// Mitsubishi GX Works2 project: ZhaoQing_HuaCheng2_1.1修改   PLC: Q03UDE
// 化成线2号柜

TYPE BarCylinderIO : STRUCT
  xPresentSwitch : BOOL;  (* 行程开关 *)
  xBarCylinder : BOOL;  (* 阻挡气缸 *)
  xEmpty : BOOL;  (* 为空指示 *)
  xTransportMotorCW : BOOL;  (* 输送电机正转 *)
  tLeaveDelay : TIME;  (* 放行延时 *)
  xUnload : BOOL;  (* 下料 *)
  xBarCylinderButton : BOOL;  (* 阻挡气缸 *)
  xTransportMotorCWButton : BOOL;  (* 输送电机正转按钮 *)
  xLoad : BOOL;  (* 上料 *)
  xNextRun : BOOL;  (* 下位设备开始运行 *)
  xTransportMotorCCWButton : BOOL;  (* 输送电机反转按钮 *)
  xTransportMotorCCW : BOOL;  (* 输送电机反转 *)
END_STRUCT END_TYPE

TYPE ConveyorIO : STRUCT
  xCWPresent : BOOL;  (* 正转检测有无传感器 *)
  xCCWPresent : BOOL;  (* 反转检测有无传感器 *)
  xLoad : BOOL;  (* 上料请求 *)
  xUnload : BOOL;  (* 下料请求 *)
  xMotorCW : BOOL;  (* 电机正转 *)
  xMotorCCW : BOOL;  (* 电机反转 *)
  xEmpty : BOOL;  (* 线体状态为空 *)
  xNextRun : BOOL;  (* 下段线体运行 *)
  xUnloadCCW : BOOL;  (* 下料为反转 *)
  xloadCCW : BOOL;  (* 上料为反转 *)
  xLeave : BOOL;  (* 已经离开 *)
  xForward : BOOL;  (* 正转手动 *)
  xBackward : BOOL;  (* 反转手动 *)
  xBusy : BOOL;  (* 工作中 *)
  tLeaveDelay : TIME;  (* 离开延时设置 *)
  xPutInto : BOOL;  (* 线体直接投入物料 *)
  xLoadAlarrm : BOOL;  (* 上料报警 *)
  xUnloadAlarm : BOOL;  (* 下料报警 *)
  tLoadDelay : TIME;  (* 进入延时设置 *)
  iProductCategory : INT;  (* 产品种类 *)
END_STRUCT END_TYPE

TYPE RGVCommunication : STRUCT
  xFullLoadRequest : BOOL;  (* 满框上料请求 *)
  xFullUnloadRequest : BOOL;  (* 满框下料请求 *)
  xEmptyLoadRequest : BOOL;  (* 空框上料请求 *)
  xEmptyUnloadRequest : BOOL;  (* 空框下料请求 *)
  xFullLoadRequestAkn : BOOL;  (* 满框上料请求确认 *)
  xFullUnloadRequestAkn : BOOL;  (* 满框下料请求确认 *)
  xEmptyLoadRequestAkn : BOOL;  (* 空框上料请求确认 *)
  xEmptyUnloadRequestAkn : BOOL;  (* 空框下料请求确认 *)
  xFullLoadComplete : BOOL;  (* 满框上料完成 *)
  xFullUnloadComplete : BOOL;  (* 满框下料完成 *)
  xEmptyLoadComplete : BOOL;  (* 空框上料完成 *)
  xEmptyUnloadComplete : BOOL;  (* 空框下料完成 *)
  xFullLoadCompleteAkn : BOOL;  (* 满框上料完成确认 *)
  xFullUnloadCompleteAkn : BOOL;  (* 满框下料完成确认 *)
  xEmptyLoadCompleteAkn : BOOL;  (* 空框上料完成确认 *)
  xEmptyUnloadCompleteAkn : BOOL;  (* 空框下料完成确认 *)
END_STRUCT END_TYPE

TYPE ShuttleCarIO : STRUCT
  xReady : BOOL;  (* 准备就绪 *)
  xForward : BOOL;  (* 正转 *)
  xBackward : BOOL;  (* 反转 *)
  iCurrentPos : INT;  (* 当前位置 *)
  iDestinationPos : INT;  (* 目标位置 *)
  xCW : BOOL;  (* 正转输出 *)
  xCCW : BOOL;  (* 反转输出 *)
  xBrake : BOOL;  (* 刹车 *)
  xHomeSwitch : BOOL;  (* 零位接近开关 *)
  xPosLimit : BOOL;  (* 正限位 *)
  xNegLimit : BOOL;  (* 负限位 *)
  xMDIExe : BOOL;  (* MDI开始 *)
  xMDIDone : BOOL;  (* MDI 完成 *)
  xPassLimit : BOOL;  (* 限位屏蔽 *)
  xPosLimitCatch : BOOL;  (* 正限位捕捉 *)
  xNegLimitCatch : BOOL;  (* 负限位捕捉 *)
  xHomeExe : BOOL;  (* 开始寻零 *)
  xHomeDone : BOOL;  (* 寻零完成 *)
  xHomeBusy : BOOL;  (* 寻零中 *)
  xHomeFailed : BOOL;  (* 寻零失败 *)
  xBusy : BOOL;  (* 工作中 *)
END_STRUCT END_TYPE

TYPE SwitchIO : STRUCT
  xLiftCylinderRetractDetect : BOOL;
  xLiftCylinderExtendDetect : BOOL;
  xLiftCylinderRetract : BOOL;
  xLiftCylinderExtend : BOOL;
  xEntryBarCylinderRetract : BOOL;
  xLiftCylinderExtendInit : BOOL;
  xEntryEnable : BOOL;
  xExitEnable : BOOL;
  xExitBarCylinderRetract : BOOL;
  xSwithEnable : BOOL;
  xLiftCylinderRetractButton : BOOL;
  xLiftCylinderExtendButton : BOOL;
  xEntryBarCylinderRetractButton : BOOL;
  xExitBarCylinderRetractButton : BOOL;
END_STRUCT END_TYPE

// global labels: Global1
VAR_GLOBAL
  g_xAuto AT M11 : BOOL;  (* 自动 *)
  g_xManual : BOOL;  (* 手动 *)
  g_xEStop AT X3 : BOOL;  (* 急停 *)
  g_xReset AT X0 : BOOL;  (* 复位 *)
  g_xStackLampRed AT Y100 : BOOL;
  g_xStackLampAmber AT Y101 : BOOL;
  g_xStackLampGreen AT Y102 : BOOL;
  g_xBuzzer AT Y103 : BOOL;
  g_xStop AT M2 : BOOL;  (* 停止 *)
  g_xLocalAutoStart AT M1 : BOOL;
  g_xRemoteAutoStart AT M0 : BOOL;
  g_xRemoteAuto AT M10 : BOOL;
  g_iState AT D40 : INT;
  g_iLocalAutoStep : INT;
  g_xError : BOOL;
  g_xStart : BOOL;  (* 启动 *)
END_VAR

// task Task_01 (event TRUE, interval 0, priority 31): Start, POU, UDP

FUNCTION_BLOCK BarCylinder
VAR_IN_OUT
  BarCylinderIO : BarCylinderIO;
END_VAR
VAR
  m_tonViaDelay : TON;  (* 卸料延时定时器 *)
  m_xViaDelay : BOOL;  (* 通过延时 *)
  m_tViaDelayElapse : TIME;  (* 通过延时当前时间 *)
  m_xInitial : BOOL;  (* 初始化 *)
END_VAR
  (***********************************************************************
阻挡器模块，
由一个行程开关，一个阻挡器，一个倍速链输送电机组成
具有手动与自动模式
xEmpty显示当前为空料的状态
xUnload为卸料信号，连接下一设备的xEmpty信号
*************************************************************************)

  (*初始化，离开延时时间设置为5秒*)
IF NOT m_xInitial THEN
	 BarCylinderIO.tLeaveDelay :=T#5s;
	m_xInitial:=1;
END_IF;
IF g_xManual THEN    (*手动*)
	BarCylinderIO.xNextRun:=0;
	IF BarCylinderIO.xBarCylinderButton THEN
		BarCylinderIO.xBarCylinder:=1;
	ELSE
		BarCylinderIO.xBarCylinder:=0;
	END_IF;
	IF BarCylinderIO.xTransportMotorCWButton 
		AND NOT BarCylinderIO.xTransportMotorCCWButton 
		AND NOT BarCylinderIO.xTransportMotorCCW   THEN
		BarCylinderIO.xTransportMotorCW:=1;
	ELSE
		BarCylinderIO.xTransportMotorCW:=0;
	END_IF;
	IF BarCylinderIO.xTransportMotorCCWButton 
		AND NOT BarCylinderIO.xTransportMotorCWButton 
		AND NOT BarCylinderIO.xTransportMotorCW   THEN
		BarCylinderIO.xTransportMotorCCW:=1;
	ELSE
		BarCylinderIO.xTransportMotorCCW:=0;
	END_IF;
END_IF;
(*离开延时定时器*)
m_tonViaDelay(IN:=NOT  BarCylinderIO.xPresentSwitch AND g_xAuto  ,PT:= BarCylinderIO.tLeaveDelay ,Q:= BarCylinderIO.xEmpty ,ET:=m_tViaDelayElapse );

IF g_xAuto THEN(*自动*)
    IF BarCylinderIO.xUnload  AND NOT BarCylinderIO.xEmpty AND NOT BarCylinderIO.xNextRun THEN(*收到卸料命令，当阻挡器不为空时*)
    	BarCylinderIO.xBarCylinder:=1;
    	BarCylinderIO.xNextRun:=1;(*确保下料命令只执行一次，防止物料在输送过程中又有卸料命令导致多事卸料*)
    	BarCylinderIO.xTransportMotorCW:=1;
    END_IF;
    IF NOT  BarCylinderIO.xUnload  THEN
    	BarCylinderIO.xNextRun:=0;
    END_IF;
    (*如果为空，气缸顶起*)
   IF  BarCylinderIO.xEmpty  THEN
   	   BarCylinderIO.xBarCylinder:=0;
   	   IF BarCylinderIO.xLoad THEN
	   	   BarCylinderIO.xTransportMotorCW:=1;
	   END_IF;
   END_IF;
   IF NOT BarCylinderIO.xUnload AND NOT  BarCylinderIO.xEmpty THEN
   	    BarCylinderIO.xTransportMotorCW:=0;
   	END_IF;
END_IF;
IF NOT g_xEStop THEN
	 BarCylinderIO.xTransportMotorCW:=0;
	 BarCylinderIO.xTransportMotorCCW:=0;
	 BarCylinderIO.xBarCylinder:=0;
END_IF;
END_FUNCTION_BLOCK

FUNCTION_BLOCK Conveyor
VAR
  tRundelay : TIME;  (* 离开延时 *)
END_VAR
VAR_IN_OUT
  ConveyorMotor : ConveyorIO;  (* 输送线输入输出 *)
END_VAR
VAR
  iStep : INT;  (* 上料步骤 *)
  m_tLoadTimer : TIME;  (* 上料计时器 *)
  m_tUnloadTimer : TIME;  (* 下料计时器 *)
  m_tonLeaveDelay : TON;  (* 离开延时定时器 *)
  m_xLeaveDelayOut : BOOL;  (* 离开延时 *)
  m_tLeaveCurrentTime : TIME;
  m_tonLoadAlarm : TON;  (* 上料延时报警 *)
END_VAR
VAR CONSTANT
  LOAD_UNLOAD_TIME : TIME := T#30s;  (* 延时报警常量 *)
END_VAR
VAR
  m_tonUnloadAlam : TON;  (* 下料报警定时器 *)
  m_tonLoadDelay : TON;  (* 离开延时定时器 *)
  m_xLoadDelayOut : BOOL;  (* 离开延时 *)
  m_tLoadCurrentTime : TIME;
  m_xInitial : BOOL;  (* 初始化 *)
END_VAR
(*////////////////////////////////////////////////////////////////////////////////////////////////////////////
//传输线控制FB块，可控制单方向线体，双向旋转线体，支持双向上下料            
//线体初始化后为空的情况下输入xLoad信号即可进行上料动作，使用xLoadCCW信号可反方向上料
//增加了产品信息和产品种类的储存，当传输线为空和上料进行标志位为零的情况下清除产品信息和产品种类
//使用方式是在置位xLoad信号后，把产品信息和产品种类传入，等下料后自动清零
//线体不为空的情况下使用xUnload信号可进行下料动作，物料有无传感器的下降沿后出发计时器，延时断开传输线旋转
//单方向传输线体把xLoadCCW、xUnloadCCW设置为零，双向线体上料方向和下料反向的,方向固定的 把xUnloadCCW设置为1
//双方向线体双向都能上下料的要根据上料的方向来设置xLoadCCW,xUnloadCCW
//增加工作中信号xBusy当电机正转 显示为工作中
//增加上下料超时报警，xLoadAlarm，xUnloadAlarm，设定时间在LOAD_UNLOAD_TIME常量上，现在设置的为30秒
//增加xPutInto信号，用于直接投入的物料，检测开关感应到后，直接进入下料流程，上升沿有效
//离开延时改为变量 iLeaveDelay 默认为0 离开检测开关离输送线尾端比较远的线体需要根据情况设定100ms为单位
增加初始化标志位，增加进入延时时间，初始化为进入延时时间为0 ，离开延时时间为2S，通过外围接口可以更改
//修改信息  修改后请增加版本
//YAO      V1.0
///////////////////////////////////////////////////////////////////////////////////////////////////////////
********************************************************)
IF NOT m_xInitial THEN
	ConveyorMotor.tLoadDelay:=T#0s;
END_IF;
m_xInitial:=1;
IF g_xAuto THEN
CASE iStep OF
	0:
	ConveyorMotor.xMotorCW:=0;
	ConveyorMotor.xMotorCCW:=0;
	ConveyorMotor.xNextRun:=0;
IF g_xEStop  THEN
	IF (ConveyorMotor.xCWPresent OR ConveyorMotor.xCCWPresent)  THEN
		iStep:=3;
		ConveyorMotor.xEmpty:=0;
		ELSE
		iStep:=1;
		ConveyorMotor.xEmpty:=1;
	END_IF;
END_IF;		
	1: 
	IF ConveyorMotor.xLoad    
		AND ConveyorMotor.xMotorCW=0   
		AND ConveyorMotor.xMotorCCW=0   
		AND ConveyorMotor.xEmpty THEN	
		iStep:=2;
	END_IF;
	2: 
	IF ConveyorMotor.xloadCCW THEN
		ConveyorMotor.xMotorCCW:=1; 
		ConveyorMotor.xMotorCW:=0;
	ELSE
	    ConveyorMotor.xMotorCW:=1;  
		ConveyorMotor.xMotorCCW:=0;
	END_IF;
		m_tonLoadDelay(IN:= (ConveyorMotor.xCWPresent AND NOT ConveyorMotor.xloadCCW) 
		                                        OR (ConveyorMotor.xCCWPresent AND ConveyorMotor.xloadCCW) ,
		                               PT:= ConveyorMotor.tLoadDelay ,
		                               Q:= m_xLoadDelayOut ,
		                               ET:= m_tLoadTimer );
	    IF m_xLoadDelayOut THEN 	 
		    iStep:=3;
		END_IF;
	3:
	ConveyorMotor.xMotorCW:=0;
	ConveyorMotor.xMotorCCW:=0;
	ConveyorMotor.xEmpty:=0;
	IF ConveyorMotor.xUnload THEN 
		iStep:=4;
	END_IF;
	4:	
	IF ConveyorMotor.xUnloadCCW THEN   
		ConveyorMotor.xMotorCCW:=1;  
		ConveyorMotor.xMotorCW:=0;
		ELSE
	    ConveyorMotor.xMotorCW:=1;  
		ConveyorMotor.xMotorCCW:=0;
	END_IF;
	ConveyorMotor.xNextRun:=1; 
	IF NOT ConveyorMotor.xUnload THEN 
		istep:=0;
	END_IF;
END_CASE;
IF LDP(TRUE,ConveyorMotor.xPutInto) THEN
	iStep:=0;
END_IF;
END_IF;
IF ConveyorMotor.xEmpty AND NOT ConveyorMotor.xLoad THEN
	ConveyorMotor.iProductCategory:=0;
END_IF;
IF g_xEStop=0 OR g_xReset THEN
	iStep:=0;
END_IF;	

IF g_xManual THEN
	iStep:=0;

	IF ConveyorMotor.xForward 
		AND ConveyorMotor.xBackward=0 
		AND ConveyorMotor.xMotorCCW=0
		AND g_xEStop THEN
		ConveyorMotor.xMotorCW:=1;
		ConveyorMotor.xMotorCCW:=0;
		ELSE
		ConveyorMotor.xMotorCW:=0;
	END_IF;

	IF ConveyorMotor.xBackward 
		AND ConveyorMotor.xForward=0 
		AND ConveyorMotor.xMotorCW=0
		AND g_xEStop  THEN
		ConveyorMotor.xMotorCCW:=1;
		conveyormotor.xMotorCW:=0;
		ELSE
		ConveyorMotor.xMotorCCW:=0;
	END_IF;
END_IF;
IF ConveyorMotor.xMotorCCW        
	OR ConveyorMotor.xMotorCW THEN  
	ConveyorMotor.xBusy:=1;
	ELSE
	ConveyorMotor.xBusy:=0;
END_IF;
m_tonLoadAlarm(IN:= iStep=2 ,PT:= LOAD_UNLOAD_TIME,Q:= ConveyorMotor.xLoadAlarrm ,ET:= m_tLoadTimer );
m_tonUnloadAlam(IN:= iStep=4,PT:= LOAD_UNLOAD_TIME,Q:= ConveyorMotor.xUnloadAlarm,ET:= m_tUnloadTimer );
END_FUNCTION_BLOCK

PROGRAM POU
VAR
  Lifter3 : ShuttleCar;
  Lifter3IO : ShuttleCarIO;
  H3000Conveyor11 : Conveyor;
  H3000Conveyor11IO : ConveyorIO;
  H3000Conveyor12 : Conveyor;
  H3000Conveyor12IO : ConveyorIO;
  H3000Conveyor13 : Conveyor;
  H3000Conveyor13IO : ConveyorIO;
  H3000Conveyor14 : Conveyor;
  H3000Conveyor14IO : ConveyorIO;
  H3000Conveyor15 : Conveyor;
  H3000Conveyor15IO : ConveyorIO;
  H3000Conveyor16 : Conveyor;
  H3000Conveyor16IO : ConveyorIO;
  H3000Conveyor17 : Conveyor;
  H3000Conveyor17IO : ConveyorIO;
  H3000Conveyor18 : Conveyor;
  H3000Conveyor18IO : ConveyorIO;
  H3000Conveyor19 : Conveyor;
  H3000Conveyor19IO : ConveyorIO;
  H3000Conveyor20 : Conveyor;
  H3000Conveyor20IO : ConveyorIO;
  H3000Conveyor21 : Conveyor;
  H3000Conveyor21IO : ConveyorIO;
  H3000Conveyor22 : Conveyor;
  H3000Conveyor22IO : ConveyorIO;
  H2200Conveyor13 : Conveyor;
  H2200Conveyor13IO : ConveyorIO;
  H2200Conveyor14 : Conveyor;
  H2200Conveyor14IO : ConveyorIO;
  H2200Conveyor15 : Conveyor;
  H2200Conveyor15IO : ConveyorIO;
  H2200Conveyor16 : Conveyor;
  H2200Conveyor16IO : ConveyorIO;
  H2200Conveyor17 : Conveyor;
  H2200Conveyor17IO : ConveyorIO;
  H2200Conveyor18 : Conveyor;
  H2200Conveyor18IO : ConveyorIO;
  H2200Conveyor19 : Conveyor;
  H2200Conveyor19IO : ConveyorIO;
  H2200Conveyor20 : Conveyor;
  H2200Conveyor20IO : ConveyorIO;
  H2200Conveyor21 : Conveyor;
  H2200Conveyor21IO : ConveyorIO;
  H2200Conveyor22 : Conveyor;
  H2200Conveyor22IO : ConveyorIO;
  H1000Conveyor11 : Conveyor;
  H1000Conveyor11IO : ConveyorIO;
  H1000Conveyor12 : Conveyor;
  H1000Conveyor12IO : ConveyorIO;
  H1000Conveyor13 : Conveyor;
  H1000Conveyor13IO : ConveyorIO;
  H1000Conveyor14 : Conveyor;
  H1000Conveyor14IO : ConveyorIO;
  H1000Conveyor15 : Conveyor;
  H1000Conveyor15IO : ConveyorIO;
  H1000Conveyor16 : Conveyor;
  H1000Conveyor16IO : ConveyorIO;
  H1000Conveyor19 : Conveyor;
  H1000Conveyor19IO : ConveyorIO;
  H1000Conveyor20 : Conveyor;
  H1000Conveyor20IO : ConveyorIO;
  Conveyor3 : Conveyor;
  Conveyor3IO : ConveyorIO;
  Lifter4 : ShuttleCar;
  Lifter4IO : ShuttleCarIO;
  Conveyor4 : Conveyor;
  Conveyor4IO : ConveyorIO;
  Lifter5 : ShuttleCar;
  Lifter5IO : ShuttleCarIO;
  Conveyor5 : Conveyor;
  Conveyor5IO : ConveyorIO;
  H850Conveyor1 : Conveyor;
  H850Conveyor1IO : ConveyorIO;
  H850Conveyor2 : Conveyor;
  H850Conveyor2IO : ConveyorIO;
  H2200Conveyor1 : Conveyor;
  H2200Conveyor1IO : ConveyorIO;
  ShuttleCar1 : ShuttleCar;
  ShuttleCar1IO : ShuttleCarIO;
  ConveyorShuttleCar : Conveyor;
  ConveyorShuttleCarIO : ConveyorIO;
  H1000Rotor1 : ShuttleCar;
  H1000Rotor1IO : ShuttleCarIO;
  H1000Rotor2 : ShuttleCar;
  H1000Rotor2IO : ShuttleCarIO;
  H1000Rotor1Cylinder : ShuttleCar;
  H1000Rotor1CylinderIO : ShuttleCarIO;
  H1000Rotor2Cylinder : ShuttleCar;
  H1000Rotor2CylinderIO : ShuttleCarIO;
  H850Conveyor1Trans : Conveyor;  (* 二封设备入口接驳 *)
  H850Conveyor1IOTrans : ConveyorIO;  (* 二封设备入口接驳 *)
  H850Conveyor2Trans : Conveyor;  (* 二封设备入口接驳 *)
  H850Conveyor2IOTrans : ConveyorIO;  (* 二封设备入口接驳 *)
  H850Conveyor3Trans : Conveyor;  (* 二封设备入口接驳 *)
  H850Conveyor3IOTrans : ConveyorIO;  (* 二封设备入口接驳 *)
  H850Conveyor4Trans : Conveyor;  (* 二封设备入口接驳 *)
  H850Conveyor4IOTrans : ConveyorIO;  (* 二封设备入口接驳 *)
  H850Conveyor5Trans : Conveyor;  (* 二封设备入口接驳 *)
  H850Conveyor5IOTrans : ConveyorIO;  (* 二封设备入口接驳 *)
  H850Conveyor6Trans : Conveyor;  (* 二封设备入口接驳 *)
  H850Conveyor6IOTrans : ConveyorIO;  (* 二封设备入口接驳 *)
  H850Conveyor7Trans : Conveyor;  (* 二封设备入口接驳 *)
  H850Conveyor7IOTrans : ConveyorIO;  (* 二封设备入口接驳 *)
  H850Conveyor8Trans : Conveyor;  (* 二封设备入口接驳 *)
  H850Conveyor8IOTrans : ConveyorIO;  (* 二封设备入口接驳 *)
  Lifter4VelocityCtl : ShuttleCarVelocityFB;
  Lifter5VelocityCtl : ShuttleCarVelocityFB;
  m_tofShuttleCar1LeaveDelay : TOF;  (* f *)
  m_xShuttleCar1LeaveDelay : BOOL;
  m_tShuttleCar1LeaveDelay : TIME;
  Lifter3VelocityCtl : ShuttleCarVelocityFB;
  H380EmptyABumperBar : BarCylinder;
  H380EmptyABumperBarIO : BarCylinderIO;
  H380EmptyBBumperBar : BarCylinder;
  H380EmptyBBumperBarIO : BarCylinderIO;
  ChemRGV : RGVCommunication;
  QuarPackageRGV : RGVCommunication;
END_VAR
(*---------我在516行加了一整行*)
Lifter3(ShuttleCarInOut:=Lifter3IO);
ShuttleCarCurrentPosition( X5A OR X5B ,X5A ,X5B, FALSE, Lifter3IO.iCurrentPos );
Lifter3VelocityCtl(xEnable:= g_xManual,xMotorCW:= Lifter3IO.xCW ,xMotorCCW:= Lifter3IO.xCCW ,
                               xPosition1Switch:= X5A ,xDecelerationSwitch:= X59 ,
	                           xPosition2Switch:=X5B ,xHighSpeed:= Y163);
Lifter3IO.xReady:=X4;
Lifter3Io.xForward:=M50;
Lifter3IO.xBackward:=M51;
Lifter3IO.xPosLimit:=X5C;
Lifter3IO.xNegLimit:=X5D;
Y161:=Lifter3IO.xCW;
Y162:=Lifter3IO.xCCW;
Y166:=Lifter3IO.xBrake;

Conveyor3(ConveyorMotor:=Conveyor3IO);
Conveyor3IO.xForward:=M52;
Conveyor3IO.xBackward:=M53;
Conveyor3IO.xCWPresent:=X61;
Conveyor3IO.xCCWPresent:=X62;
Y168:=Conveyor3IO.xMotorCW;
Y167:=Conveyor3IO.xMotorCCW;
Conveyor3IO.xUnloadCCW:=1;

Lifter4(ShuttleCarInOut:=Lifter4IO);
ShuttleCarCurrentPosition( X64 OR X65 ,X64 ,X65, FALSE, Lifter4IO.iCurrentPos );
Lifter4VelocityCtl(xEnable:= g_xAuto,xMotorCW:= Lifter4IO.xCW ,xMotorCCW:= Lifter4IO.xCCW ,
                               xPosition1Switch:= X64 ,xDecelerationSwitch:= X63 ,
	                           xPosition2Switch:=X65 ,xHighSpeed:= Y16B);
Lifter4IO.xReady:=X5;
Lifter4Io.xForward:=M54;
Lifter4IO.xBackward:=M55;
Lifter4IO.xPosLimit:=X66;
Lifter4IO.xNegLimit:=X67;
Y169:=Lifter4IO.xCW;
Y16A:=Lifter4IO.xCCW;
Y16E:=Lifter4IO.xBrake;

Conveyor4(ConveyorMotor:=Conveyor4IO);
Conveyor4IO.xForward:=M56;
Conveyor4IO.xBackward:=M57;
Conveyor4IO.xCWPresent:=X6B;
Conveyor4IO.xCCWPresent:=X6C;
Y170:=Conveyor4IO.xMotorCW;
Y16F:=Conveyor4IO.xMotorCCW;
Conveyor4IO.xUnloadCCW:=1;

Lifter5(ShuttleCarInOut:=Lifter5IO);
ShuttleCarCurrentPosition( X6E OR X6F ,X6E ,X6F, FALSE, Lifter5IO.iCurrentPos );
Lifter5VelocityCtl(xEnable:= g_xAuto,
                               xMotorCW:= Lifter5IO.xCW ,
                               xMotorCCW:= Lifter5IO.xCCW,
                               xPosition1Switch:=X6E,
                               xDecelerationSwitch:= X6D,
	                           xPosition2Switch:=X6F,
	                           xHighSpeed:= Y173 );
Lifter5IO.xReady:=X6;
Lifter5Io.xForward:=M58;
Lifter5IO.xBackward:=M59;
Lifter5IO.xPosLimit:=X70;
Lifter5IO.xNegLimit:=X71;
Y171:=Lifter5IO.xCW;
Y172:=Lifter5IO.xCCW;
Y176:=Lifter5IO.xBrake;

Conveyor5(ConveyorMotor:=Conveyor5IO);
Conveyor5IO.xForward:=M60;
Conveyor5IO.xBackward:=M61;
Conveyor5IO.xCWPresent:=X75;
Conveyor5IO.xCCWPresent:=X76;
Y178:=Conveyor5IO.xMotorCW;
Y177:=Conveyor5IO.xMotorCCW;
Conveyor5IO.xUnloadCCW:=1;

ShuttleCar1(ShuttleCarInOut:=ShuttleCar1IO);
ShuttleCarCurrentPosition(( NOT X53 AND NOT X54) OR (NOT X53 AND NOT X55) OR (NOT X54 AND NOT  X55) ,
                                                       NOT X53 AND NOT X54 ,
                                                       NOT X53 AND NOT X55,
                                                       NOT X54 AND NOT  X55, 
                                                       ShuttleCar1IO.iCurrentPos );
ShuttleCar1IO.xReady:=X7;
ShuttleCar1IO.xForward:=M62;
ShuttleCar1IO.xBackward:=M63;
ShuttleCar1IO.xPosLimit:=X51;
ShuttleCar1IO.xNegLimit:=X52;
Y1AB:=ShuttleCar1IO.xCW;
Y1AC:=ShuttleCar1IO.xCCW;
Y12B:=ShuttleCar1IO.xBrake;

ConveyorShuttleCar(ConveyorMotor:=ConveyorShuttleCarIO);
ConveyorShuttleCarIO.xForward:=M64;
ConveyorShuttleCarIO.xBackward:=M65;
ConveyorShuttleCarIO.xCWPresent:=X56;
ConveyorShuttleCarIO.xCCWPresent:=X57;
Y153:=ConveyorShuttleCarIO.xMotorCW;
Y154:=ConveyorShuttleCarIO.xMotorCCW;

H3000Conveyor11(ConveyorMotor:=H3000Conveyor11IO);
H3000Conveyor11IO.xForward:=M30;
H3000Conveyor11IO.xCWPresent:=X8;
Y108:=H3000Conveyor11IO.xMotorCW;

H3000Conveyor12(ConveyorMotor:=H3000Conveyor12IO);
H3000Conveyor12IO.xForward:=M31;
H3000Conveyor12IO.xCWPresent:=X9;
Y109:=H3000Conveyor12IO.xMotorCW;

H3000Conveyor13(ConveyorMotor:=H3000Conveyor13IO);
H3000Conveyor13IO.xForward:=M32;
H3000Conveyor13IO.xCWPresent:=XA;
Y10A:=H3000Conveyor13IO.xMotorCW;

H3000Conveyor14(ConveyorMotor:=H3000Conveyor14IO);
H3000Conveyor14IO.xForward:=M33;
H3000Conveyor14IO.xCWPresent:=XB;
Y10B:=H3000Conveyor14IO.xMotorCW;

H3000Conveyor15(ConveyorMotor:=H3000Conveyor15IO);
H3000Conveyor15IO.xForward:=M34;
H3000Conveyor15IO.xCWPresent:=XC;
Y10C:=H3000Conveyor15IO.xMotorCW;

H3000Conveyor16(ConveyorMotor:=H3000Conveyor16IO);
H3000Conveyor16IO.xForward:=M34;
H3000Conveyor16IO.xCWPresent:=XD;
Y10D:=H3000Conveyor16IO.xMotorCW;

H3000Conveyor17(ConveyorMotor:=H3000Conveyor17IO);
H3000Conveyor17IO.xForward:=M35;
H3000Conveyor17IO.xCWPresent:=XE;
Y10E:=H3000Conveyor17IO.xMotorCW;

H3000Conveyor18(ConveyorMotor:=H3000Conveyor18IO);
H3000Conveyor18IO.xForward:=M36;
H3000Conveyor18IO.xCWPresent:=XF;
Y10F:=H3000Conveyor18IO.xMotorCW;

H3000Conveyor19(ConveyorMotor:=H3000Conveyor19IO);
H3000Conveyor19IO.xForward:=M37;
H3000Conveyor19IO.xCWPresent:=X10;
Y110:=H3000Conveyor19IO.xMotorCW;

H3000Conveyor20(ConveyorMotor:=H3000Conveyor20IO);
H3000Conveyor20IO.xForward:=M38;
H3000Conveyor20IO.xCWPresent:=X11;
Y111:=H3000Conveyor20IO.xMotorCW;

H3000Conveyor21(ConveyorMotor:=H3000Conveyor21IO);
H3000Conveyor21IO.xForward:=M39;
H3000Conveyor21IO.xCWPresent:=X12;
Y112:=H3000Conveyor21IO.xMotorCW;

H3000Conveyor22(ConveyorMotor:=H3000Conveyor22IO);
H3000Conveyor22IO.xForward:=M40;
H3000Conveyor22IO.xCWPresent:=X13;
Y113:=H3000Conveyor22IO.xMotorCW;

H850Conveyor1(ConveyorMotor:=H850Conveyor1IO);
H850Conveyor1IO.xForward:=M41;
H850Conveyor1IO.xCWPresent:=X4E;
Y14E:=H850Conveyor1IO.xMotorCW;

H850Conveyor2(ConveyorMotor:=H850Conveyor2IO);
H850Conveyor2IO.xForward:=M42;
H850Conveyor2IO.xCWPresent:=X4F;
Y14F:=H850Conveyor2IO.xMotorCW;

H2200Conveyor1(ConveyorMotor:=H2200Conveyor1IO);
H2200Conveyor1IO.xForward:=M43;
H2200Conveyor1IO.xCWPresent:=X4D;
Y14D:=H2200Conveyor1IO.xMotorCW;



H2200Conveyor13(ConveyorMotor:=H2200Conveyor13IO);
H2200Conveyor13IO.xForward:=M44;
H2200Conveyor13IO.xCWPresent:=X2F;
Y12F:=H2200Conveyor13IO.xMotorCW;

H2200Conveyor14(ConveyorMotor:=H2200Conveyor14IO);
H2200Conveyor14IO.xForward:=M45;
H2200Conveyor14IO.xCWPresent:=X30;
Y130:=H2200Conveyor14IO.xMotorCW;

H2200Conveyor15(ConveyorMotor:=H2200Conveyor15IO);
H2200Conveyor15IO.xForward:=M46;
H2200Conveyor15IO.xCWPresent:=X31;
Y131:=H2200Conveyor15IO.xMotorCW;

H2200Conveyor16(ConveyorMotor:=H2200Conveyor16IO);
H2200Conveyor16IO.xForward:=M47;
H2200Conveyor16IO.xCWPresent:=X32;
Y132:=H2200Conveyor16IO.xMotorCW;

H2200Conveyor17(ConveyorMotor:=H2200Conveyor17IO);
H2200Conveyor17IO.xForward:=M48;
H2200Conveyor17IO.xCWPresent:=X33;
Y133:=H2200Conveyor17IO.xMotorCW;

H2200Conveyor18(ConveyorMotor:=H2200Conveyor18IO);
H2200Conveyor18IO.xForward:=M49;
H2200Conveyor18IO.xCWPresent:=X34;
Y134:=H2200Conveyor18IO.xMotorCW;

H2200Conveyor19(ConveyorMotor:=H2200Conveyor19IO);
H2200Conveyor19IO.xForward:=M70;
H2200Conveyor19IO.xCWPresent:=X35;
Y135:=H2200Conveyor19IO.xMotorCW;

H2200Conveyor20(ConveyorMotor:=H2200Conveyor20IO);
H2200Conveyor20IO.xForward:=M71;
H2200Conveyor20IO.xCWPresent:=X36;
Y136:=H2200Conveyor20IO.xMotorCW;

H2200Conveyor21(ConveyorMotor:=H2200Conveyor21IO);
H2200Conveyor21IO.xForward:=M72;
H2200Conveyor21IO.xCWPresent:=X37;
Y137:=H2200Conveyor21IO.xMotorCW;

H2200Conveyor22(ConveyorMotor:=H2200Conveyor22IO);
H2200Conveyor22IO.xForward:=M73;
H2200Conveyor22IO.xCWPresent:=X38;
Y138:=H2200Conveyor22IO.xMotorCW;

H1000Conveyor11(ConveyorMotor:=H1000Conveyor11IO);
H1000Conveyor11IO.xForward:=M75;
H1000Conveyor11IO.xCWPresent:=X3A;
Y13A:=H1000Conveyor11IO.xMotorCW;

H1000Conveyor12(ConveyorMotor:=H1000Conveyor12IO);
H1000Conveyor12IO.xForward:=M76;
H1000Conveyor12IO.xCWPresent:=X3B;
Y13B:=H1000Conveyor12IO.xMotorCW;

H1000Conveyor13(ConveyorMotor:=H1000Conveyor13IO);
H1000Conveyor13IO.xForward:=M77;
H1000Conveyor13IO.xCWPresent:=X3C;
Y13C:=H1000Conveyor13IO.xMotorCW;

H1000Conveyor14(ConveyorMotor:=H1000Conveyor14IO);
H1000Conveyor14IO.xForward:=M78;
H1000Conveyor14IO.xCWPresent:=X3D;
Y13D:=H1000Conveyor14IO.xMotorCW;

H1000Conveyor15(ConveyorMotor:=H1000Conveyor15IO);
H1000Conveyor15IO.xForward:=M79;
H1000Conveyor15IO.xCWPresent:=X3E;
Y13E:=H1000Conveyor15IO.xMotorCW;

H1000Rotor2(ShuttleCarInOut:=H1000Rotor2IO);
ShuttleCarCurrentPosition( X9F OR X9E ,X9F ,X9E, FALSE, H1000Rotor2IO.iCurrentPos );
H1000Rotor2IO.xReady:=TRUE;
H1000Rotor2IO.xForward:=M93;
H1000Rotor2IO.xBackward:=M94;
H1000Rotor2IO.xPosLimit:=XB0;
H1000Rotor2IO.xNegLimit:=XB1;
Y1BC:=H1000Rotor2IO.xCW;
Y1BD:=H1000Rotor2IO.xCCW;
Y12A:=H1000Rotor2IO.xBrake;

H1000Rotor2Cylinder(ShuttleCarInOut:=H1000Rotor2CylinderIO);
ShuttleCarCurrentPosition( XA0 OR XA1 ,XA1 ,XA0, FALSE, H1000Rotor2CylinderIO.iCurrentPos );
H1000Rotor2CylinderIO.xReady:=TRUE;
H1000Rotor2CylinderIO.xForward:=M87;
H1000Rotor2CylinderIO.xBackward:=M88;
H1000Rotor2CylinderIO.xPosLimit:=TRUE;
H1000Rotor2CylinderIO.xNegLimit:=TRUE;
Y1A1:=H1000Rotor2CylinderIO.xCW;
Y1A0:=H1000Rotor2CylinderIO.xCCW;

H1000Conveyor16(ConveyorMotor:=H1000Conveyor16IO);
H1000Conveyor16IO.xForward:=M80;
H1000Conveyor16IO.xCWPresent:=X3F;
Y13F:=H1000Conveyor16IO.xMotorCW;

H1000Rotor1(ShuttleCarInOut:=H1000Rotor1IO);
ShuttleCarCurrentPosition( X9A OR X9B ,X9A ,X9B, FALSE, H1000Rotor1IO.iCurrentPos );
H1000Rotor1IO.xReady:=TRUE;
H1000Rotor1IO.xForward:=M83;
H1000Rotor1IO.xBackward:=M84;
H1000Rotor1IO.xPosLimit:=X99;
H1000Rotor1IO.xNegLimit:=X98;
Y104:=H1000Rotor1IO.xCW;
Y105:=H1000Rotor1IO.xCCW;
Y129:=H1000Rotor1IO.xBrake;

H1000Rotor1Cylinder(ShuttleCarInOut:=H1000Rotor1CylinderIO);
ShuttleCarCurrentPosition( X9D OR X9C ,X9D ,X9C, FALSE, H1000Rotor1CylinderIO.iCurrentPos );
H1000Rotor1CylinderIO.xReady:=TRUE;
H1000Rotor1CylinderIO.xForward:=M85;
H1000Rotor1CylinderIO.xBackward:=M86;
H1000Rotor1CylinderIO.xPosLimit:=TRUE;
H1000Rotor1CylinderIO.xNegLimit:=TRUE;
Y19C:=H1000Rotor1CylinderIO.xCW;
Y19B:=H1000Rotor1CylinderIO.xCCW;

H1000Conveyor19(ConveyorMotor:=H1000Conveyor19IO);
H1000Conveyor19IO.tLeaveDelay:=t#10s;
H1000Conveyor19IO.xForward:=M81;
H1000Conveyor19IO.xCWPresent:=X42;
Y142:=H1000Conveyor19IO.xMotorCW;

H1000Conveyor20(ConveyorMotor:=H1000Conveyor20IO);
H1000Conveyor20IO.xForward:=M82;
H1000Conveyor20IO.xCWPresent:=X43;
Y143:=H1000Conveyor20IO.xMotorCW;

H850Conveyor1Trans(ConveyorMotor:=H850Conveyor1IOTrans);
H850Conveyor1IOTrans.xForward:=M120;
H850Conveyor1IOTrans.xCWPresent:=XA3;
Y1A3:=H850Conveyor1IOTrans.xMotorCW;

H850Conveyor2Trans(ConveyorMotor:=H850Conveyor2IOTrans);
H850Conveyor2IOTrans.xForward:=M121;
H850Conveyor2IOTrans.xCWPresent:=XA4;
Y1A4:=H850Conveyor2IOTrans.xMotorCW;

H850Conveyor3Trans(ConveyorMotor:=H850Conveyor3IOTrans);
H850Conveyor3IOTrans.xForward:=M122;
H850Conveyor3IOTrans.xCWPresent:=XA5;
Y1A5:=H850Conveyor3IOTrans.xMotorCW;

H850Conveyor4Trans(ConveyorMotor:=H850Conveyor4IOTrans);
H850Conveyor4IOTrans.xForward:=M123;
H850Conveyor4IOTrans.xCWPresent:=XA6;
Y1A6:=H850Conveyor4IOTrans.xMotorCW;

H850Conveyor5Trans(ConveyorMotor:=H850Conveyor5IOTrans);
H850Conveyor5IOTrans.xForward:=M124;
H850Conveyor5IOTrans.xCWPresent:=XA7;
Y1A7:=H850Conveyor5IOTrans.xMotorCW;

H850Conveyor6Trans(ConveyorMotor:=H850Conveyor6IOTrans);
H850Conveyor6IOTrans.xForward:=M125;
H850Conveyor6IOTrans.xCWPresent:=XA8;
Y1A8:=H850Conveyor6IOTrans.xMotorCW;

H850Conveyor7Trans(ConveyorMotor:=H850Conveyor7IOTrans);
H850Conveyor7IOTrans.xForward:=M126;
H850Conveyor7IOTrans.xCWPresent:=XA9;
Y1A9:=H850Conveyor7IOTrans.xMotorCW;

H850Conveyor8Trans(ConveyorMotor:=H850Conveyor8IOTrans);
H850Conveyor8IOTrans.xForward:=M127;
H850Conveyor8IOTrans.xCWPresent:=XAA;
Y1AA:=H850Conveyor8IOTrans.xMotorCW;

H380EmptyABumperBar(BarCylinderIO:= H380EmptyABumperBarIO);
H380EmptyABumperBarIO.xBarCylinderButton:=M68;
H380EmptyABumperBarIO.xTransportMotorCWButton:=M89;
H380EmptyABumperBarIO.xTransportMotorCCWButton:=M90;
H380EmptyABumperBarIO.xPresentSwitch:=X49;
Y149:=H380EmptyABumperBarIO.xBarCylinder;
Y15E:=H380EmptyABumperBarIO.xTransportMotorCW;
Y15D:=H380EmptyABumperBarIO.xTransportMotorCCW;

H380EmptyBBumperBar(BarCylinderIO:= H380EmptyBBumperBarIO);
H380EmptyBBumperBarIO.xBarCylinderButton:=M69;
H380EmptyBBumperBarIO.xTransportMotorCWButton:=M91;
H380EmptyBBumperBarIO.xTransportMotorCCWButton:=M92;
H380EmptyBBumperBarIO.xPresentSwitch:=X4A;
Y14A:=H380EmptyBBumperBarIO.xBarCylinder;
Y15F:=H380EmptyBBumperBarIO.xTransportMotorCW;
Y160:=H380EmptyBBumperBarIO.xTransportMotorCCW;

(*自动状态*)
IF g_xAuto THEN
	(********3000线体满框去二封************)
	D201.0:=H3000Conveyor11IO.xEmpty;
	H3000Conveyor11IO.xLoad:=D401.0;
	H3000Conveyor11IO.xUnload:=H3000Conveyor12IO.xEmpty;
	H3000Conveyor12IO.xLoad:=H3000Conveyor11IO.xNextRun;
	H3000Conveyor12IO.xUnload:=H3000Conveyor13IO.xEmpty;
	H3000Conveyor13IO.xLoad:=H3000Conveyor12IO.xNextRun;	
	H3000Conveyor13IO.xUnload:=H3000Conveyor14IO.xEmpty;
	H3000Conveyor14IO.xLoad:=H3000Conveyor13IO.xNextRun;
	H3000Conveyor14IO.xUnload:=H3000Conveyor15IO.xEmpty;
	H3000Conveyor15IO.xLoad:=H3000Conveyor14IO.xNextRun;
	H3000Conveyor15IO.xUnload:=H3000Conveyor16IO.xEmpty;
	H3000Conveyor16IO.xLoad:=H3000Conveyor15IO.xNextRun;
	H3000Conveyor16IO.xUnload:=H3000Conveyor17IO.xEmpty;
	H3000Conveyor17IO.xLoad:=H3000Conveyor16IO.xNextRun;
	H3000Conveyor17IO.xUnload:=H3000Conveyor18IO.xEmpty;
	H3000Conveyor18IO.xLoad:=H3000Conveyor17IO.xNextRun;	
	H3000Conveyor18IO.xUnload:=H3000Conveyor19IO.xEmpty;
	H3000Conveyor19IO.xLoad:=H3000Conveyor18IO.xNextRun;	
	H3000Conveyor19IO.xUnload:=H3000Conveyor20IO.xEmpty;
	H3000Conveyor20IO.xLoad:=H3000Conveyor19IO.xNextRun;
	H3000Conveyor20IO.xUnload:=H3000Conveyor21IO.xEmpty;
	H3000Conveyor21IO.xLoad:=H3000Conveyor20IO.xNextRun;
	H3000Conveyor21IO.xUnload:=H3000Conveyor22IO.xEmpty;
	H3000Conveyor22IO.xLoad:=H3000Conveyor21IO.xNextRun;
		(********3000线体满框去二封提升机************)
	IF Lifter5IO.iCurrentPos=2 AND X6F  THEN
		H3000Conveyor22IO.xUnload:=Conveyor5IO.xEmpty;
	ELSE
		H3000Conveyor22IO.xUnload:=0;		
	END_IF;
	conveyor5Io.xLoad:=H3000Conveyor22Io.xNextRun;
	IF Conveyor5IO.xEmpty  THEN
		Lifter5IO.xMDIExe:=1;
		Lifter5IO.iDestinationPos:=2;
	END_IF;
	IF Conveyor5IO.xEmpty=0 THEN
		Lifter5io.xMDIExe:=1;
		Lifter5IO.iDestinationPos:=1;
	END_IF;
	IF ldp(TRUE,Conveyor5IO.xEmpty=0) THEN
		D10:=D10+1;
	END_IF;
	IF  M74 THEN
	D10:=0;
	END_IF;
IF  Lifter5IO.iCurrentPos=1 AND X6E  THEN
	Conveyor5IO.xUnload:=H850Conveyor2IO.xEmpty;
ELSE
	Conveyor5IO.xUnload:=0;
END_IF;
	H850Conveyor2IO.xLoad:=Conveyor5IO.xNextRun;
	H850Conveyor2IO.xPutInto:=M881;(*临时程序*)
   (********3000线体满框去二封AGV接料************)
   H850Conveyor2IO.xUnload:=QuarPackageRGV.xFullLoadRequest;
   QuarPackageRGV.xFullLoadRequestAkn:=H850Conveyor2IO.xNextRun;
   
   (********二封AGV空框返回************)
   H850Conveyor1IO.xLoad:=QuarPackageRGV.xEmptyUnloadRequest;
   QuarPackageRGV.xEmptyUnloadRequestAkn:=H850Conveyor1IO.xNextRun;
	(********二封空框返回************)
    H850Conveyor1IO.xLoad:=M880;
    IF Conveyor4IO.xEmpty THEN
    	Lifter4Io.xMDIExe:=1;
    	Lifter4Io.iDestinationPos:=1;
    END_IF;
    IF Lifter4IO.iCurrentPos=1 AND X64   THEN
    	H850Conveyor1IO.xUnload:=Conveyor4Io.xEmpty;
    ELSE
    	H850Conveyor1IO.xUnload:=0;
    END_IF;
       Conveyor4IO.xLoad:=H850Conveyor1IO.xNextRun;
       IF Conveyor4IO.xEmpty =0 AND Lifter4IO.iCurrentPos=1  THEN
       	   Lifter4IO.xMDIExe:=1;
       	   Lifter4IO.iDestinationPos:=2;
       END_IF;
       IF Lifter4IO.iCurrentPos=2 AND  X65   THEN
       	  Conveyor4IO.xUnload:=H2200Conveyor1IO.xEmpty;
       ELSE
       	 Conveyor4IO.xUnload:=0;
       END_IF;
       H2200Conveyor1IO.xLoad:=conveyor4IO.xNextRun;
       Y158:=1; (********第一段空框A返回倍速链************)
       Y15A:=1; (********第二段空框B返回倍速链************)
   (********穿梭小车接空框************)
    IF ShuttleCar1IO.iCurrentPos=1 AND (NOT X53 AND NOT X54 ) THEN
        H2200Conveyor1IO.xUnload:=ConveyorShuttleCarIO.xEmpty;
    ELSE
    	H2200Conveyor1IO.xUnload:=0;
       	END_IF;
       	ConveyorShuttleCarIO.xLoad:= H2200Conveyor1IO.xNextRun;
      IF ConveyorShuttleCarIO.xEmpty   THEN
        ShuttleCar1IO.xMDIExe:=1;
       	ShuttleCar1IO.iDestinationPos:=1;
      END_IF;     	
      (*M882空框回流A框与B框选择，触摸屏上按钮*)
       IF ConveyorShuttleCarIO.xEmpty =0 AND NOT  M882   THEN
       	ShuttleCar1IO.xMDIExe:=1;
       	ShuttleCar1IO.iDestinationPos:=2;
       END_IF;
        IF ConveyorShuttleCarIO.xEmpty =0 AND  M882   THEN
       	ShuttleCar1IO.xMDIExe:=1;
       	ShuttleCar1IO.iDestinationPos:=3;
       END_IF;      
       	    IF (ShuttleCar1IO.iCurrentPos=2 AND NOT X53 AND NOT X55) 
       	    	OR (ShuttleCar1IO.iCurrentPos=3 AND  NOT X54 AND NOT X55 )  THEN
       	    	m_tofShuttleCar1LeaveDelay(IN:=ConveyorShuttleCarIO.xCWPresent ,PT:= T#5s ,Q:= m_xShuttleCar1LeaveDelay ,ET:= m_tShuttleCar1LeaveDelay );
       		    ConveyorShuttleCarIO.xUnload:= m_xShuttleCar1LeaveDelay;
       	    ELSE
       	        ConveyorShuttleCarIO.xUnload:=0;
       		END_IF;
    (********H2200满框去化成***********)  
    D201.1:=  H2200Conveyor13IO.xEmpty;
	H2200Conveyor13IO.xLoad:=D401.1;
	H2200Conveyor13IO.xUnload:=H2200Conveyor14IO.xEmpty;
	H2200Conveyor14IO.xLoad:=H2200Conveyor13IO.xNextRun;
	H2200Conveyor14IO.xUnload:=H2200Conveyor15IO.xEmpty;
	H2200Conveyor15IO.xLoad:=H2200Conveyor14IO.xNextRun;	
	H2200Conveyor15IO.xUnload:=H2200Conveyor16IO.xEmpty;
	H2200Conveyor16IO.xLoad:=H2200Conveyor15IO.xNextRun;	
	H2200Conveyor16IO.xUnload:=H2200Conveyor17IO.xEmpty;
	H2200Conveyor17IO.xLoad:=H2200Conveyor16IO.xNextRun;	
	H2200Conveyor17IO.xUnload:=H2200Conveyor18IO.xEmpty;
	H2200Conveyor18IO.xLoad:=H2200Conveyor17IO.xNextRun;	
	H2200Conveyor18IO.xUnload:=H2200Conveyor19IO.xEmpty;
	H2200Conveyor19IO.xLoad:=H2200Conveyor18IO.xNextRun;		
	H2200Conveyor19IO.xUnload:=H2200Conveyor20IO.xEmpty;
	H2200Conveyor20IO.xLoad:=H2200Conveyor19IO.xNextRun;		
	H2200Conveyor20IO.xUnload:=H2200Conveyor21IO.xEmpty;
	H2200Conveyor21IO.xLoad:=H2200Conveyor20IO.xNextRun;		
	H2200Conveyor21IO.xUnload:=H2200Conveyor22IO.xEmpty;
	H2200Conveyor22IO.xLoad:=H2200Conveyor21IO.xNextRun;		
    IF conveyor3IO.xEmpty THEN
    	Lifter3IO.xMDIExe:=1;
    	Lifter3IO.iDestinationPos:=2;
    END_IF;
    IF conveyor3Io.xEmpty=0 THEN
      	Lifter3IO.xMDIExe:=1;
    	Lifter3IO.iDestinationPos:=1;  	
    END_IF;
    IF Lifter3IO.iCurrentPos=2 AND X5B THEN
    	H2200Conveyor22io.xUnload:= Conveyor3io.xEmpty;
    ELSE
    	H2200Conveyor22io.xUnload:=0;
    END_IF;
    Conveyor3IO.xLoad:=H2200Conveyor22io.xNextRun;
    IF Lifter3IO.iCurrentPos=1 AND X5A THEN
    	 Conveyor3IO.xUnload:=H1000Conveyor20IO.xEmpty;
    ELSE
    	 Conveyor3IO.xUnload:=0;
    END_IF;
    	H1000Conveyor20IO.xLoad:=Conveyor3IO.xNextRun;
    	H1000Conveyor20IO.xUnload:=H1000Conveyor19IO.xEmpty;
       H1000Conveyor19IO.xLoad:=H1000Conveyor20IO.xNextRun;
      H1000Conveyor19IO.xPutInto:=SM413;                (*-----这里我加了个随时判断19conveyor的东西，暂时用*)
       (*化成RGV接料程序*)
       H1000Conveyor19IO.xUnload:=ChemRGV.xFullLoadRequest;
       ChemRGV.xFullLoadRequestAkn:=H1000Conveyor19IO.xNextRun;
       (*化成RGV空框上料程序，A缓存线——》化成*)
       H380EmptyABumperBarIO.xLoad:=ChemRGV.xEmptyLoadRequest;
 	   ChemRGV.xEmptyLoadRequestAkn:=	H380EmptyABumperBarIO.xEmpty;
        (*化成RGV空框出料程序,化成——》A缓存线*)
       H380EmptyABumperBarIO.xTransportMotorCCW:=ChemRGV.xEmptyUnloadRequest;
        ChemRGV.xEmptyUnloadRequestAkn:=H380EmptyABumperBarIO.xEmpty;          
          
        (*化成RGV满框出料程序*)
        ChemRGV.xFullUnloadRequestAkn:=H1000Conveyor16IO.xEmpty;
        H1000Conveyor16IO.xLoad:=ChemRGV.xFullUnloadRequest OR X2C ;(*----加了个按钮*)
       H1000Conveyor16IO.xUnload:=H1000Conveyor15IO.xEmpty;
       H1000Conveyor15IO.xLoad:=H1000Conveyor16IO.xNextRun ;
        H1000Conveyor15IO.xUnload:=H1000Conveyor14IO.xEmpty;
       H1000Conveyor14IO.xLoad:=H1000Conveyor15IO.xNextRun;      
         H1000Conveyor14IO.xUnload:=H1000Conveyor13IO.xEmpty;
       H1000Conveyor13IO.xLoad:=H1000Conveyor14IO.xNextRun; 
        H1000Conveyor13IO.xUnload:=H1000Conveyor12IO.xEmpty;
       H1000Conveyor12IO.xLoad:=H1000Conveyor13IO.xNextRun;
        H1000Conveyor13IO.xUnload:=H1000Conveyor12IO.xEmpty;
       H1000Conveyor12IO.xLoad:=H1000Conveyor13IO.xNextRun;
        H1000Conveyor12IO.xUnload:=H1000Conveyor11IO.xEmpty;
       H1000Conveyor11IO.xLoad:=H1000Conveyor12IO.xNextRun;      
      H1000Conveyor11IO.xUnload:=D401.2;(*接收给化成1号柜*线体10为空信号*)
      D201.2:=    H1000Conveyor11IO.xNextRun;(*发送给化成1号柜*线体10为开始旋转信号*)
END_IF;

IF g_xManual OR  g_xReset THEN
	D201:=0;
	Lifter3IO.xMDIExe:=0;
	Lifter4IO.xMDIExe:=0;
	Lifter5IO.xMDIExe:=0;
	Conveyor3IO.xLoad:=0;
	Conveyor3IO.xUnload:=0;
	Conveyor4IO.xLoad:=0;
	Conveyor4IO.xUnload:=0;
	Conveyor5IO.xLoad:=0;
	Conveyor5IO.xUnload:=0;	
	ShuttleCar1IO.xMDIExe:=0;
	ConveyorShuttleCarIO.xLoad:=0;
	ConveyorShuttleCarIO.xUnload:=0;
	IF M66 AND g_xEStop  THEN (*空框A返回倍速链 手动*)
		 Y158:=1;(*空框A返回倍速链*)
	ELSE
		Y158:=0;;(*空框A返回倍速链*)
	END_IF;
	IF M67 AND g_xEStop THEN (*空框B返回倍速链 手动*)
		 Y15A:=1;(*空框B返回倍速链*)
	ELSE
		Y15A:=0;(*空框B返回倍速链*)
	END_IF;	

	IF M91 AND NOT M92 AND NOT Y160 AND g_xEStop THEN(*化成空框B缓存倍速链手动正转*)
		Y15F:=1;(*化成空框B缓存倍速链正转*)
	ELSE
		Y15F:=0;
	END_IF;
	IF M92 AND NOT M91 AND NOT Y15F AND g_xEStop THEN(*化成空框B缓存倍速链手动反转*)
		Y160:=1;(*化成空框B缓存倍速链反转*)
	ELSE
		Y160:=0;
	END_IF;
	
	
END_IF;
END_PROGRAM

FUNCTION_BLOCK ShuttleCar
VAR_IN_OUT
  ShuttleCarInOut : ShuttleCarIO;
END_VAR
VAR
  m_xBrakeDelay : BOOL;  (* 刹车延时标志位 *)
  diCurrentPosRetain : DINT;
  m_tonBrakeDelay : TON;  (* 延时 *)
  m_tBrakeDelay : TIME;
  m_xBrake : BOOL;
  m_tBrakeDelayCurrentTime : TIME;
END_VAR
(*******************************************************************
输送小车程序，可用于使用认址片控制位置的输送车程序，可用于控制提升机，
使用了限位捕捉程序防止小车惯性过大冲过限位后继续行走，捕捉程序采用反
转复位，这样设计有弊端可能反转复位后车的位置并没有回到限位以内,当两个
限位同时碰到的时候，会使运料小车进入死锁状态，通过xPassLimit来解开死锁，
可以在触摸屏中使用一个带权限的按钮来进行控制，配合ShuttleCarCurrentPos
函数来计算位置信息
增加自动开始后将当前位置置为零的信号防止设备停在两个位置开关的中间
修改信息  修改后请增加版本
YAO      V1.0
********************************************************************)

ShuttleCarInOut.xPosLimitCatch:=LDF(TRUE,ShuttleCarInOut.xPosLimit) OR ShuttleCarInOut.xPosLimitCatch;
IF ShuttleCarInOut.xCCW THEN  
	ShuttleCarInOut.xPosLimitCatch:=0;
END_IF;

ShuttleCarInOut.xNegLimitCatch:=LDF(TRUE,ShuttleCarInOut.xNegLimit) OR ShuttleCarInOut.xNegLimitCatch;
IF ShuttleCarInOut.xCW THEN   
	ShuttleCarInOut.xNegLimitCatch:=0;  
END_IF;
IF ShuttleCarInOut.xPassLimit OR
	(ShuttleCarInOut.xNegLimitCatch 
	AND ShuttleCarInOut.xPosLimitCatch)  THEN  
	ShuttleCarInOut.xNegLimitCatch:=0; 
	ShuttleCarInOut.xPosLimitCatch:=0;
END_IF;

IF ShuttleCarInOut.xReady THEN	
    IF g_xManual THEN  
	    IF ShuttleCarInOut.xForward 
			AND ShuttleCarInOut.xBackward=0 
			AND ShuttleCarInOut.xCCW=0 
			AND ShuttleCarInOut.xPosLimitCatch=0 
			AND g_xEStop THEN
		    ShuttleCarInOut.xCW:=1;
		    ELSE
		    ShuttleCarInOut.xCW:=0;
	    END_IF;
	    IF ShuttleCarInOut.xBackward 
			AND ShuttleCarInOut.xForward=0 
			AND ShuttleCarInOut.xCW=0 
			AND ShuttleCarInOut.xNegLimitCatch=0 
			AND G_xEStop THEN  
		    ShuttleCarInOut.xCCW:=1;
		    ELSE
		    ShuttleCarInOut.xCCW:=0;
	    END_IF;
    END_IF;
  IF g_xAuto AND g_xEStop THEN  
	  IF ShuttleCarInOut.xMDIExe AND ShuttleCarInOut.iDestinationPos<>0 THEN
	
	    IF ShuttleCarInOut.iCurrentPos<ShuttleCarInOut.iDestinationPos AND ShuttleCarInOut.xPosLimitCatch=0 THEN
			ShuttleCarInOut.xCW:=1;
			ShuttleCarInOut.xCCW:=0;
			ShuttleCarInOut.xMDIDone:=0;
		END_IF;

		IF ShuttleCarInOut.iCurrentPos>ShuttleCarInOut.iDestinationPos AND ShuttleCarInOut.xNegLimitCatch=0 THEN
			ShuttleCarInOut.xCCW:=1;
			ShuttleCarInOut.xCW:=0;
			ShuttleCarInOut.xMDIDone:=0;
		END_IF;
	
		IF ShuttleCarInOut.iCurrentPos=ShuttleCarInOut.iDestinationPos THEN
			ShuttleCarInOut.xCW:=0;
			ShuttleCarInOut.xCCW:=0;
			ShuttleCarInOut.xMDIDone:=1;
			ELSE
			ShuttleCarInOut.xMDIDone:=0;
		END_IF;

		IF ShuttleCarInOut.xPosLimitCatch THEN
			ShuttleCarInOut.xCW:=0;
			ShuttleCarInOut.xMDIDone:=0;
		END_IF;

		IF ShuttleCarInOut.xNegLimitCatch THEN
			ShuttleCarInOut.xCCW:=0;
			ShuttleCarInOut.xMDIDone:=0;
		END_IF;
		ELSE
		ShuttleCarInOut.xCW:=0;
		ShuttleCarInOut.xCCW:=0;
		ShuttleCarInOut.xMDIDone:=0;
	  END_IF;
	END_IF;
	ELSE
		ShuttleCarInOut.xCW:=0;
		ShuttleCarInOut.xCCW:=0;	
END_IF;
m_tonBrakeDelay(IN:=m_xBrakeDelay ,PT:= T#100ms,Q:=m_xBrake ,ET:= m_tBrakeDelayCurrentTime);
IF (ShuttleCarInOut.xCW OR ShuttleCarInOut.xCCW) AND ShuttleCarInOut.xReady=1 THEN
	ShuttleCarInOut.xBrake:=m_xBrake;
	m_xBrakeDelay:=1;
	ELSE
	ShuttleCarInOut.xBrake:=0;
	m_xBrakeDelay:=0;
END_IF;

IF g_xEStop =0 THEN
	ShuttleCarInOut.xCW :=0;
	ShuttleCarInOut.xCCW:=0;
END_IF;

(*IF SM402 THEN 
	ShuttleCarInOut.diCurrentPos:=diCurrentPosRetain;
	ELSE
	diCurrentPosRetain:=ShuttleCarInOut.diCurrentPos;
END_IF;*)
(*自动上电后把当前位置清零，防止穿梭车不在开关位置*)
IF LDP(TRUE,g_xAuto) THEN
	ShuttleCarInOut.iCurrentPos:=0;
END_IF;
IF ShuttleCarInOut.xCW OR ShuttleCarInOut.xCCW THEN
	ShuttleCarInOut.xBusy:=1;
	ELSE
	ShuttleCarInout.xBusy:=0;
END_IF;
END_FUNCTION_BLOCK

FUNCTION ShuttleCarCurrentPosition
VAR_INPUT
  xPosition1 : BOOL;
  xPosition2 : BOOL;
  xPosition3 : BOOL;
END_VAR
(************************************
计算输送车当前位置的函数
**************************************)
IF xPosition1 THEN
	ShuttleCarCurrentPosition:=1;
END_IF;
IF xPosition2 THEN
	ShuttleCarCurrentPosition:=2;
END_IF;
IF xPosition3 THEN
	ShuttleCarCurrentPosition:=3;
END_IF;
END_FUNCTION

FUNCTION_BLOCK ShuttleCarVelocityFB
VAR_INPUT
  xEnable : BOOL;  (* 使能 *)
  xMotorCW : BOOL;  (* 电机正转 *)
  xMotorCCW : BOOL;  (* 电机反转 *)
  xPosition1Switch : BOOL;  (* 位置1开关 *)
  xDecelerationSwitch : BOOL;  (* 减速开关 *)
  xPosition2Switch : BOOL;  (* 位置2开关 *)
END_VAR
VAR
  iFloor : INT;  (* 层数 *)
END_VAR
VAR_OUTPUT
  xHighSpeed : BOOL;
END_VAR
IF xEnable THEN
	(*电机旋转，并且在位置开关上的时候触发加速*)
	IF( LDP(TRUE,xMotorCW) AND xPosition1Switch ) OR (  LDP(TRUE,xMotorCCW) AND xPosition2Switch) THEN
		xHighSpeed:=1;
		iFloor:=0;
	END_IF;
	IF LDF(TRUE,xMotorCW) OR LDF(TRUE,xMotorCCW) THEN
		xHighSpeed:=0;
    END_IF;
	IF LDP(TRUE,xDecelerationSwitch) THEN
		iFloor:=iFloor+1;
	END_IF;
	IF iFloor=2 THEN
		xHighSpeed:=0;
		iFloor:=0;
	END_IF;
ELSE
    xHighSpeed:=0;
END_IF;
END_FUNCTION_BLOCK

PROGRAM Start
IF g_xReset THEN
	SM50:=1;
ELSE
	SM50:=0;
END_IF;
CASE g_iState OF
	0: 
		g_xManual:=1;
		g_xAuto:=0;	
		g_xStackLampAmber:=1;
		g_xStackLampGreen:=0;
		g_xRemoteAuto:=0;
	1:
		g_xManual:=0;
		g_xAuto:=1;
		g_xStackLampGreen:=1;
		g_xStackLampAmber:=0;
		g_xRemoteAuto:=0;
	2:	
        g_xRemoteAuto:=1;
        g_xStackLampGreen:=1;
        g_xStackLampAmber:=0;
        g_xAuto:=0;
		g_xManual:=0;
END_CASE;
IF g_xLocalAutoStart THEN  
	g_iState:=1;
END_IF;

IF g_xStop OR g_xEStop=0 THEN 
	g_iState:=0;
END_IF;
IF g_xRemoteAutoStart THEN
	g_iState:=2;
END_IF;
END_PROGRAM

PROGRAM UDP
D200:=k2;
SP_SOCCINF( LDP(TRUE,SD1082.0) , "U0" , K1 , D110 ,D120);
SP_SOCSND( SM413 AND SD1082.0 , "U0" , K1 , D100, D200, M102 );
SP_SOCRCV( NOT M102 AND SD1082.0 , "U0" , K1, D300 , D400 ,M104 );
IF NOT SD1082.0 THEN
	D400:=0;
	D401:=0;
END_IF;
END_PROGRAM
